PROGRAM PRG_AdsClientTests
VAR
	InitDone : BOOL;
	
END_VAR

IF NOT GVL_AdsClientTests.IsRunning THEN
	MEMSET(ADR(GVL_Write.StandardTypes), 0, SIZEOF(GVL_Write.StandardTypes));
	MEMSET(ADR(GVL_Write.StandardTypes), 0, SIZEOF(GVL_Write.StandardArrays));
	MEMSET(ADR(GVL_Write.ComplexTypes), 0, SIZEOF(GVL_Write.ComplexTypes));
	MEMSET(ADR(GVL_Write.ComplexArrayTypes), 0, SIZEOF(GVL_Write.ComplexArrayTypes));
	MEMSET(ADR(GVL_Write.SpecialTypes), 0, SIZEOF(GVL_Write.SpecialTypes));
	MEMSET(ADR(GVL_Write.IssueSpecificTypes), 0, SIZEOF(GVL_Write.IssueSpecificTypes));
	
	GVL_Write.ComplexTypes.POINTER_ := ADR(GVL_Write.StandardTypes);
	GVL_Write.ComplexTypes.REFERENCE_ ref= GVL_Write.StandardTypes;
	
	GVL_AdsClientTests.IsRunning := TRUE;
END_IF

PRG_Subscription();

END_PROGRAM

(* stored: Version 1.1.0.1, ProductVersion 3.1.4024.12
   POU PRG_AdsClientTests: Id {d3e9ca6d-84a0-4f3a-9bdc-c7b060ad3f7f}, SpecialFunc None *)
